FUNCTION_BLOCK TEST_SERVICE
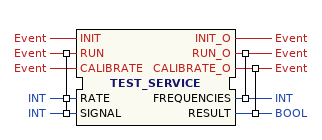
  EVENT_INPUT
    INIT;
    RUN WITH RATE, SIGNAL; {SET_ATTRIBUTE(OpcUa, Method)}
    CALIBRATE; {SET_ATTRIBUTE(OpcUa, Method)}
  END_EVENT
  EVENT_OUTPUT
    INIT_O;
    RUN_O WITH FREQUENCIES;
    CALIBRATE_O WITH RESULT;
  END_EVENT
  VAR_INPUT
    RATE : INT; {SET_ATTRIBUTE(OpcUa, Constant.RUN)}
    SIGNAL : INT; {SET_ATTRIBUTE(OpcUa, Variable.RUN)}
  END_VAR
  VAR_OUTPUT
    FREQUENCIES : INT; {SET_ATTRIBUTE(OpcUa, Variable.RUN)}
    RESULT : BOOL; {SET_ATTRIBUTE(OpcUa, CALIBRATE)}
  END_VAR
END_FUNCTION_BLOCK
(* other elements stored in the file *)
(* SelfDescription FBType=SERVICE *)
